// TIA Portal V16 export
// export: Created 2023-03-29T11:03:42.035458Z, ExportSetting WithDefaults, DisplayName Totally Integrated Automation Portal, DisplayVersion V16 Update 6, DisplayName TIA Portal Version Control Interface, DisplayVersion V16 Update 2, DisplayName TIA Portal Openness, DisplayVersion V16 Update 6, DisplayName STEP 7 Professional, DisplayVersion V16 Update 6, DisplayName STEP 7 Safety, DisplayVersion V16, DisplayName WinCC Advanced, DisplayVersion V16 Update 6
DATA_BLOCK "AI_Scalowani_Położenia_Z10_DB"   // DB33
AUTHOR : rtecmer
VERSION : 0.1
// stored: AutoNumber true, DBAccessibleFromOPCUA true, InstanceOfName AI_Scalowani_Położenia_Z10, InstanceOfType FB
"AI_Scalowani_Położenia_Z10"
   // VAR_INPUT
   //    actAI_położenie_Z10 { ExternalAccessible := 'False'; ExternalVisible := 'False'; ExternalWritable := 'False'} : Word;
   // END_VAR
   // VAR_OUTPUT
   //    isPosition : Bool;
   // END_VAR
BEGIN
END_DATA_BLOCK
